Universal Robots PolyScope program: test1.urp

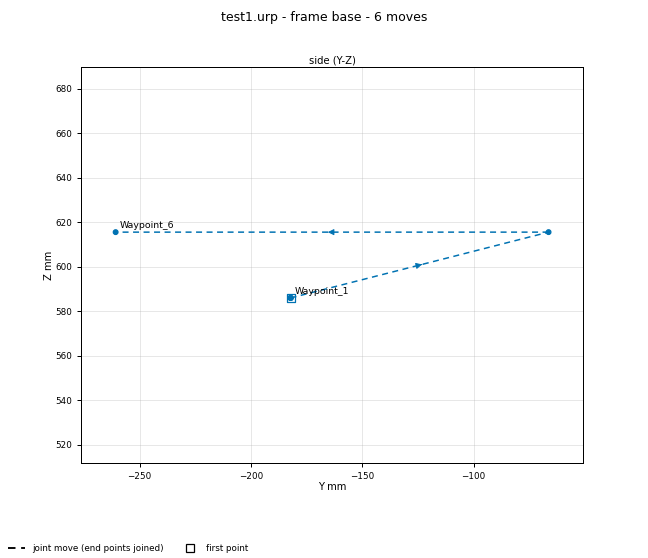
[picture p0: tool path of test1.urp in frame base, 6 of 6 moves have a stored position in this frame; points joined in program order, loops and branches not executed]
Program test1 (installation=default directory=/programs/usbdisk createdIn=5.11.10.1010502 lastSavedIn=5.11.10.1010502 robotSerialNumber=20225201339)
Calibrated DH parameters: a=[-0.000118, -0.339742, -0.555336, 0.000027, 0.000053, 0]; d=[0.180691, -465.540026, 499.223902, -33.510242, 0.119749, 0.115686]; alpha=[1.571428, -0.001093, 0.003977, 1.569316, -1.571413, 0]; deltaTheta=[0, 0.982125, 5.537749, -0.236695, 0, 0]
Robot Program (runOnlyOnce=true)
  MoveJ speed 60 deg/s, acceleration 80 deg/s^2 (useActiveTCP=true) feature=Base
    Waypoint Waypoint_1: TCP in base x=-603.932 y=-182.199 z=585.988 mm, rx=1.0808 ry=-1.1846 rz=-1.325 rad; joints [-1.388, -50.293, 40.85, 2.74, -86.412, -0.037] deg; TCP offset x=-0.188 y=3.576 z=256.261 mm, rx=-0.0017 ry=3.1416 rz=0 rad
    Waypoint Waypoint_2: motionParameters(nextMotionTime=5); TCP in base x=-603.932 y=-182.182 z=585.984 mm, rx=0.8199 ry=-1.4532 rz=-1.5211 rad; joints [-9.256, -56.241, 50.955, -1.145, -73.81, -4.017] deg
    Waypoint Waypoint_3: motionParameters(nextMotionTime=5); TCP in base x=-603.927 y=-182.226 z=585.983 mm, rx=1.2789 ry=-0.798 rz=-0.7446 rad; joints [12.246, -49.007, 38.982, 3.406, -109.321, -8.011] deg
    Waypoint Waypoint_4: motionParameters(nextMotionTime=5); TCP in base x=-603.935 y=-182.23 z=585.959 mm, rx=1.027 ry=-0.9699 rz=-1.2971 rad; joints [1.506, -51.547, 37.36, -1.697, -91.097, 0.082] deg
    Waypoint Waypoint_5: motionParameters(nextMotionTime=5); TCP in base x=-603.926 y=-66.335 z=615.534 mm, rx=1.0269 ry=-0.9698 rz=-1.2971 rad; joints [-5.42, -52.954, 36.657, 0.247, -97.766, -1.832] deg
    Waypoint Waypoint_6: motionParameters(nextMotionTime=5); TCP in base x=-603.917 y=-260.811 z=615.53 mm, rx=1.0956 ry=-0.9183 rz=-1.3508 rad; joints [6.618, -46.209, 25.142, 5.483, -87.601, 6.407] deg
